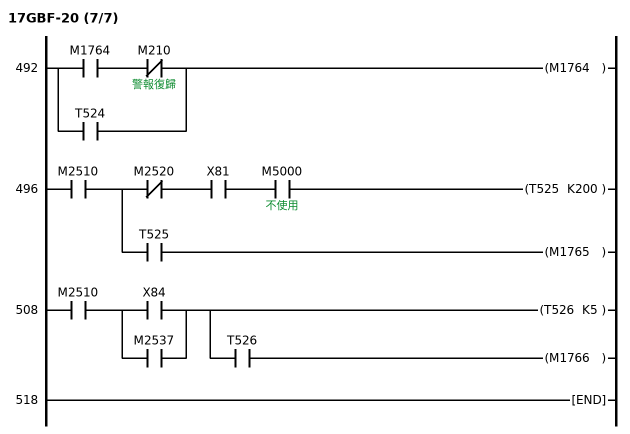
[picture p96: ladder of 17GBF-20, rungs at steps 492 to 518]
492   LD      M1764
      ANI     M210  ; 警報復歸
      OR      T524
      OUT     M1764
496   LD      M2510
      MPS
      ANI     M2520
      AND     X81
      AND     M5000  ; 不使用
      OUT     T525 K200
      MPP
      AND     T525
      OUT     M1765
508   LD      M2510
      LD      X84
      OR      M2537
      ANB
      OUT     T526 K5
      AND     T526
      OUT     M1766
518   END
END_PROGRAM

PROGRAM 18GCV
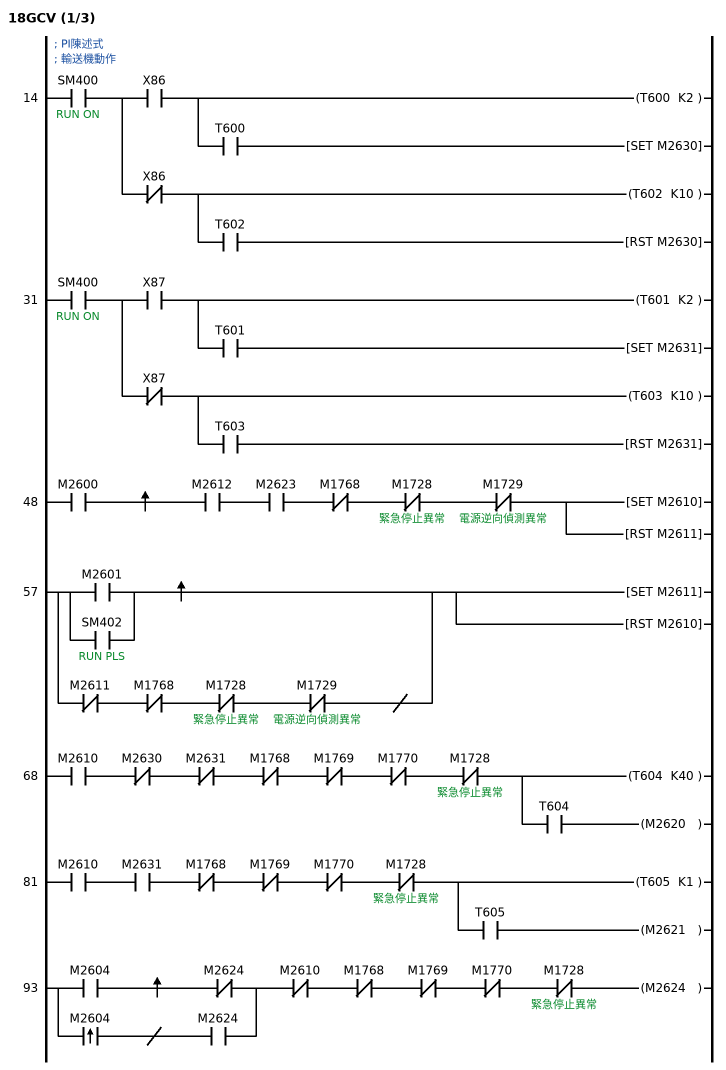
; PI陳述式
; 輸送機動作
14    LD      SM400  ; RUN ON
      MPS
      AND     X86
      OUT     T600 K2
      AND     T600
      SET     M2630
      MPP
      ANI     X86
      OUT     T602 K10
      AND     T602
      RST     M2630
31    LD      SM400  ; RUN ON
      MPS
      AND     X87
      OUT     T601 K2
      AND     T601
      SET     M2631
      MPP
      ANI     X87
      OUT     T603 K10
      AND     T603
      RST     M2631
48    LD      M2600
      MEP
      AND     M2612
      AND     M2623
      ANI     M1768
      ANI     M1728  ; 緊急停止異常
      ANI     M1729  ; 電源逆向偵測異常
      SET     M2610
      RST     M2611
57    LD      M2601
      OR      SM402  ; RUN PLS
      MEP
      LDI     M2611
      ANI     M1768
      ANI     M1728  ; 緊急停止異常
      ANI     M1729  ; 電源逆向偵測異常
      INV
      ORB
      SET     M2611
      RST     M2610
68    LD      M2610
      ANI     M2630
      ANI     M2631
      ANI     M1768
      ANI     M1769
      ANI     M1770
      ANI     M1728  ; 緊急停止異常
      OUT     T604 K40
      AND     T604
      OUT     M2620
81    LD      M2610
      AND     M2631
      ANI     M1768
      ANI     M1769
      ANI     M1770
      ANI     M1728  ; 緊急停止異常
      OUT     T605 K1
      AND     T605
      OUT     M2621
93    LD      M2604
      MEP
      ANI     M2624
      LDP     M2604
      INV
      AND     M2624
      ORB
      ANI     M2610
      ANI     M1768
      ANI     M1769
      ANI     M1770
      ANI     M1728  ; 緊急停止異常
      OUT     M2624
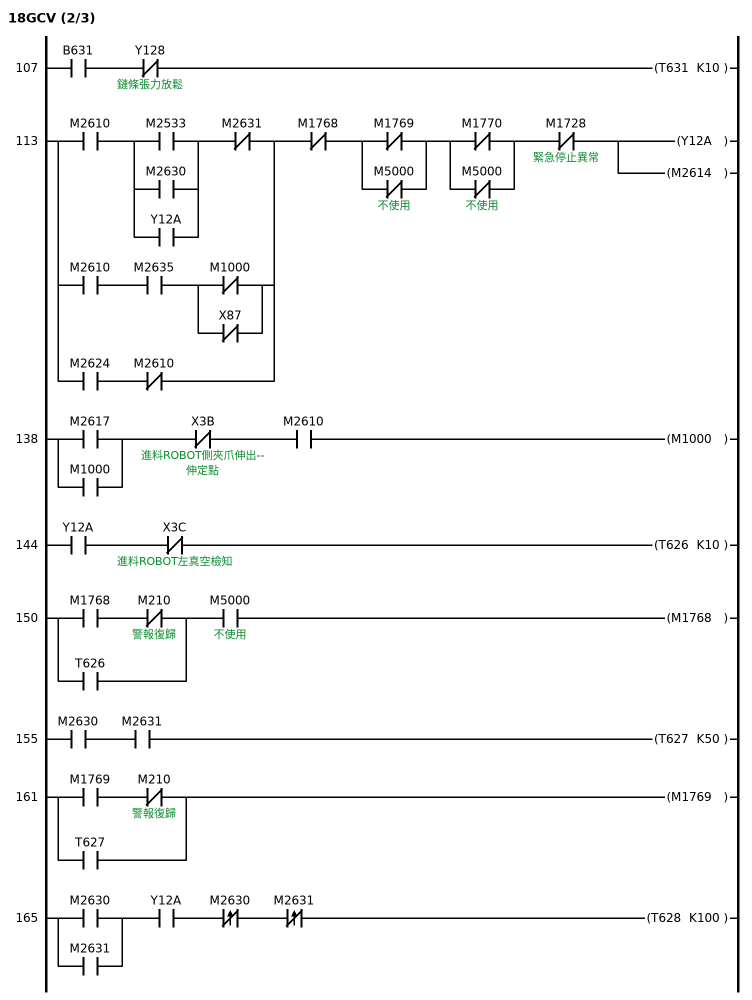
107   LD      B631
      ANI     Y128  ; 鏈條張力放鬆
      OUT     T631 K10
113   LD      M2610
      LD      M2533
      OR      M2630
      OR      Y12A
      ANB
      ANI     M2631
      LD      M2610
      AND     M2635
      LDI     M1000
      ORI     X87
      ANB
      ORB
      LD      M2624
      ANI     M2610
      ORB
      ANI     M1768
      LDI     M1769
      ORI     M5000  ; 不使用
      ANB
      LDI     M1770
      ORI     M5000  ; 不使用
      ANB
      ANI     M1728  ; 緊急停止異常
      OUT     Y12A
      OUT     M2614
138   LD      M2617
      OR      M1000
      ANI     X3B  ; 進料ROBOT側夾爪伸出--伸定點
      AND     M2610
      OUT     M1000
144   LD      Y12A
      ANI     X3C  ; 進料ROBOT左真空檢知
      OUT     T626 K10
150   LD      M1768
      ANI     M210  ; 警報復歸
      OR      T626
      AND     M5000  ; 不使用
      OUT     M1768
155   LD      M2630
      AND     M2631
      OUT     T627 K50
161   LD      M1769
      ANI     M210  ; 警報復歸
      OR      T627
      OUT     M1769
165   LD      M2630
      OR      M2631
      AND     Y12A
      ANDPI   M2630
      ANDPI   M2631
      OUT     T628 K100
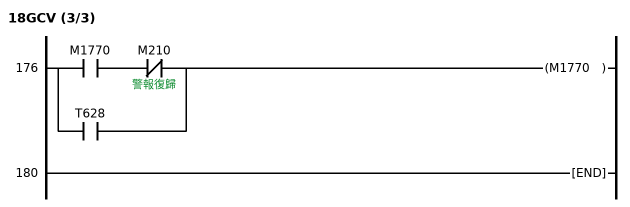
176   LD      M1770
      ANI     M210  ; 警報復歸
      OR      T628
      OUT     M1770
180   END
END_PROGRAM

PROGRAM 19GTC-7
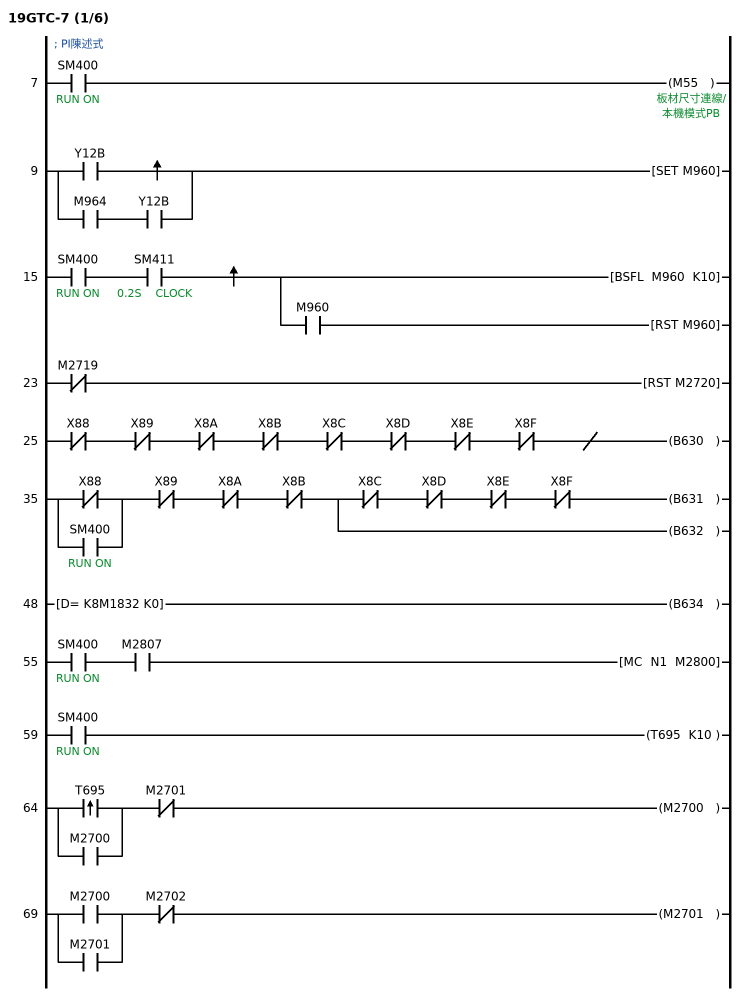
; PI陳述式
7     LD      SM400  ; RUN ON
      OUT     M55  ; 板材尺寸連線/本機模式PB
9     LD      Y12B
      MEP
      LD      M964
      AND     Y12B
      ORB
      SET     M960
15    LD      SM400  ; RUN ON
      AND     SM411  ; 0.2S    CLOCK
      MEP
      BSFL    M960 K10
      AND     M960
      RST     M960
23    LDI     M2719
      RST     M2720
25    LDI     X88
      ANI     X89
      ANI     X8A
      ANI     X8B
      ANI     X8C
      ANI     X8D
      ANI     X8E
      ANI     X8F
      INV
      OUT     B630
35    LDI     X88
      OR      SM400  ; RUN ON
      ANI     X89
      ANI     X8A
      ANI     X8B
      MPS
      ANI     X8C
      ANI     X8D
      ANI     X8E
      ANI     X8F
      OUT     B631
      MPP
      OUT     B632
48    LDD=    K8M1832 K0
      OUT     B634
55    LD      SM400  ; RUN ON
      AND     M2807
      MC      N1 M2800
59    LD      SM400  ; RUN ON
      OUT     T695 K10
64    LDP     T695
      OR      M2700
      ANI     M2701
      OUT     M2700
69    LD      M2700
      OR      M2701
      ANI     M2702
      OUT     M2701
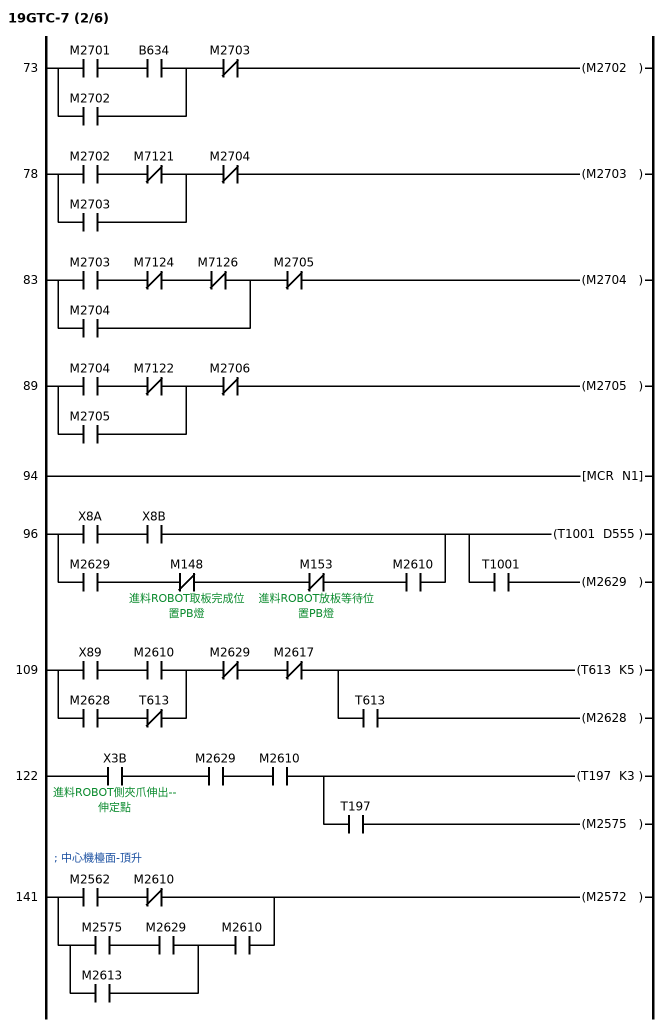
73    LD      M2701
      AND     B634
      OR      M2702
      ANI     M2703
      OUT     M2702
78    LD      M2702
      ANI     M7121
      OR      M2703
      ANI     M2704
      OUT     M2703
83    LD      M2703
      ANI     M7124
      ANI     M7126
      OR      M2704
      ANI     M2705
      OUT     M2704
89    LD      M2704
      ANI     M7122
      OR      M2705
      ANI     M2706
      OUT     M2705
94    MCR     N1
96    LD      X8A
      AND     X8B
      LD      M2629
      ANI     M148  ; 進料ROBOT取板完成位置PB燈
      ANI     M153  ; 進料ROBOT放板等待位置PB燈
      AND     M2610
      ORB
      OUT     T1001 D555
      AND     T1001
      OUT     M2629
109   LD      X89
      AND     M2610
      LD      M2628
      ANI     T613
      ORB
      ANI     M2629
      ANI     M2617
      OUT     T613 K5
      AND     T613
      OUT     M2628
122   LD      X3B  ; 進料ROBOT側夾爪伸出--伸定點
      AND     M2629
      AND     M2610
      OUT     T197 K3
      AND     T197
      OUT     M2575
; 中心機檯面-頂升
141   LD      M2562
      ANI     M2610
      LD      M2575
      AND     M2629
      OR      M2613
      AND     M2610
      ORB
      OUT     M2572
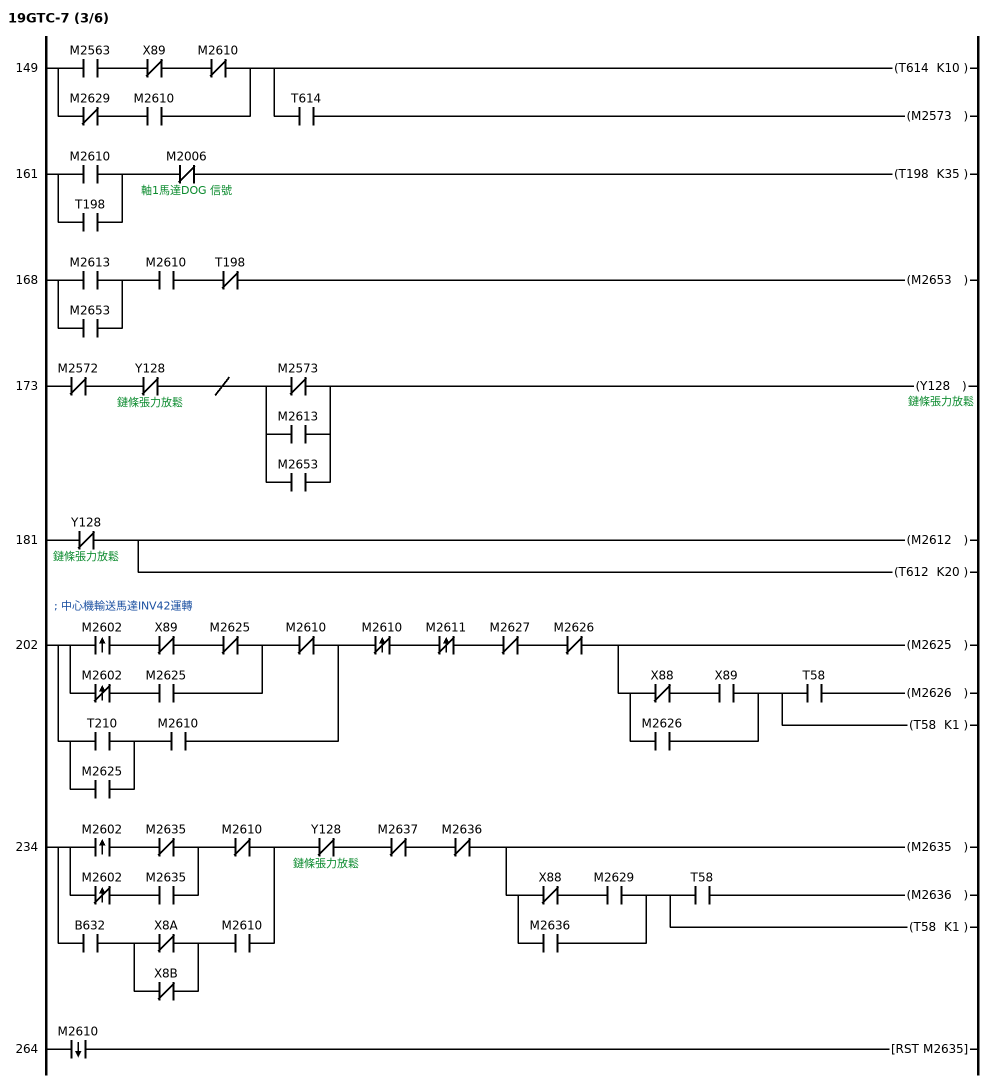
149   LD      M2563
      ANI     X89
      ANI     M2610
      LDI     M2629
      AND     M2610
      ORB
      OUT     T614 K10
      AND     T614
      OUT     M2573
161   LD      M2610
      OR      T198
      ANI     M2006  ; 軸1馬達DOG 信號
      OUT     T198 K35
168   LD      M2613
      OR      M2653
      AND     M2610
      ANI     T198
      OUT     M2653
173   LDI     M2572
      ANI     Y128  ; 鏈條張力放鬆
      INV
      LDI     M2573
      OR      M2613
      OR      M2653
      ANB
      OUT     Y128  ; 鏈條張力放鬆
181   LDI     Y128  ; 鏈條張力放鬆
      OUT     M2612
      OUT     T612 K20
; 中心機輸送馬達INV42運轉
202   LDP     M2602
      ANI     X89
      ANI     M2625
      LDPI    M2602
      AND     M2625
      ORB
      ANI     M2610
      LD      T210
      OR      M2625
      AND     M2610
      ORB
      ANDPI   M2610
      ANDPI   M2611
      ANI     M2627
      ANI     M2626
      OUT     M2625
      LDI     X88
      AND     X89
      OR      M2626
      ANB
      MPS
      AND     T58
      OUT     M2626
      MPP
      OUT     T58 K1
234   LDP     M2602
      ANI     M2635
      LDPI    M2602
      AND     M2635
      ORB
      ANI     M2610
      LD      B632
      LDI     X8A
      ORI     X8B
      ANB
      AND     M2610
      ORB
      ANI     Y128  ; 鏈條張力放鬆
      ANI     M2637
      ANI     M2636
      OUT     M2635
      LDI     X88
      AND     M2629
      OR      M2636
      ANB
      MPS
      AND     T58
      OUT     M2636
      MPP
      OUT     T58 K1
264   LDF     M2610
      RST     M2635
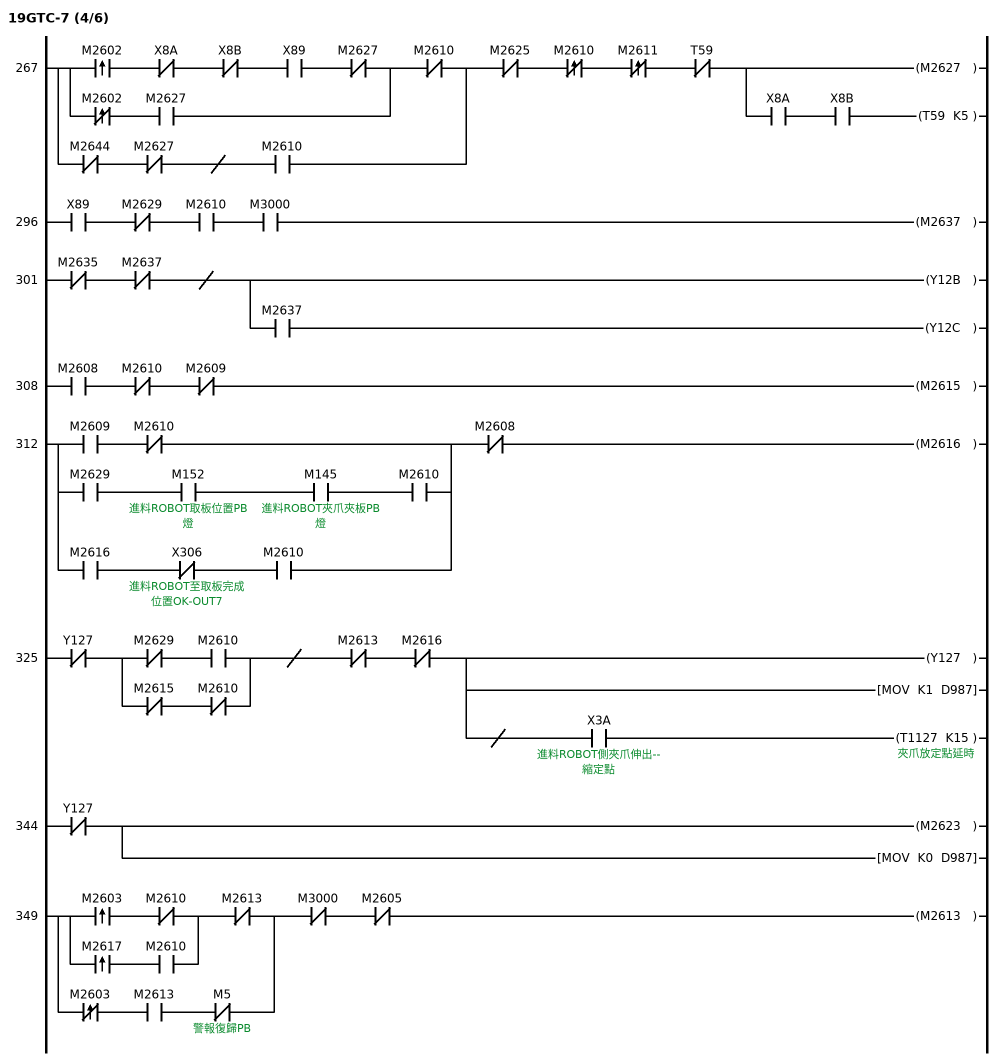
267   LDP     M2602
      ANI     X8A
      ANI     X8B
      AND     X89
      ANI     M2627
      LDPI    M2602
      AND     M2627
      ORB
      ANI     M2610
      LDI     M2644
      ANI     M2627
      INV
      AND     M2610
      ORB
      ANI     M2625
      ANDPI   M2610
      ANDPI   M2611
      ANI     T59
      OUT     M2627
      AND     X8A
      AND     X8B
      OUT     T59 K5
296   LD      X89
      ANI     M2629
      AND     M2610
      AND     M3000
      OUT     M2637
301   LDI     M2635
      ANI     M2637
      INV
      OUT     Y12B
      AND     M2637
      OUT     Y12C
308   LD      M2608
      ANI     M2610
      ANI     M2609
      OUT     M2615
312   LD      M2609
      ANI     M2610
      LD      M2629
      AND     M152  ; 進料ROBOT取板位置PB燈
      AND     M145  ; 進料ROBOT夾爪夾板PB燈
      AND     M2610
      ORB
      LD      M2616
      ANI     X306  ; 進料ROBOT至取板完成位置OK-OUT7
      AND     M2610
      ORB
      ANI     M2608
      OUT     M2616
325   LDI     Y127
      LDI     M2629
      AND     M2610
      LDI     M2615
      ANI     M2610
      ORB
      ANB
      INV
      ANI     M2613
      ANI     M2616
      OUT     Y127
      MOV     K1 D987
      INV
      AND     X3A  ; 進料ROBOT側夾爪伸出--縮定點
      OUT     T1127 K15  ; 夾爪放定點延時
344   LDI     Y127
      OUT     M2623
      MOV     K0 D987
349   LDP     M2603
      ANI     M2610
      LDP     M2617
      AND     M2610
      ORB
      ANI     M2613
      LDPI    M2603
      AND     M2613
      ANI     M5  ; 警報復歸PB
      ORB
      ANI     M3000
      ANI     M2605
      OUT     M2613
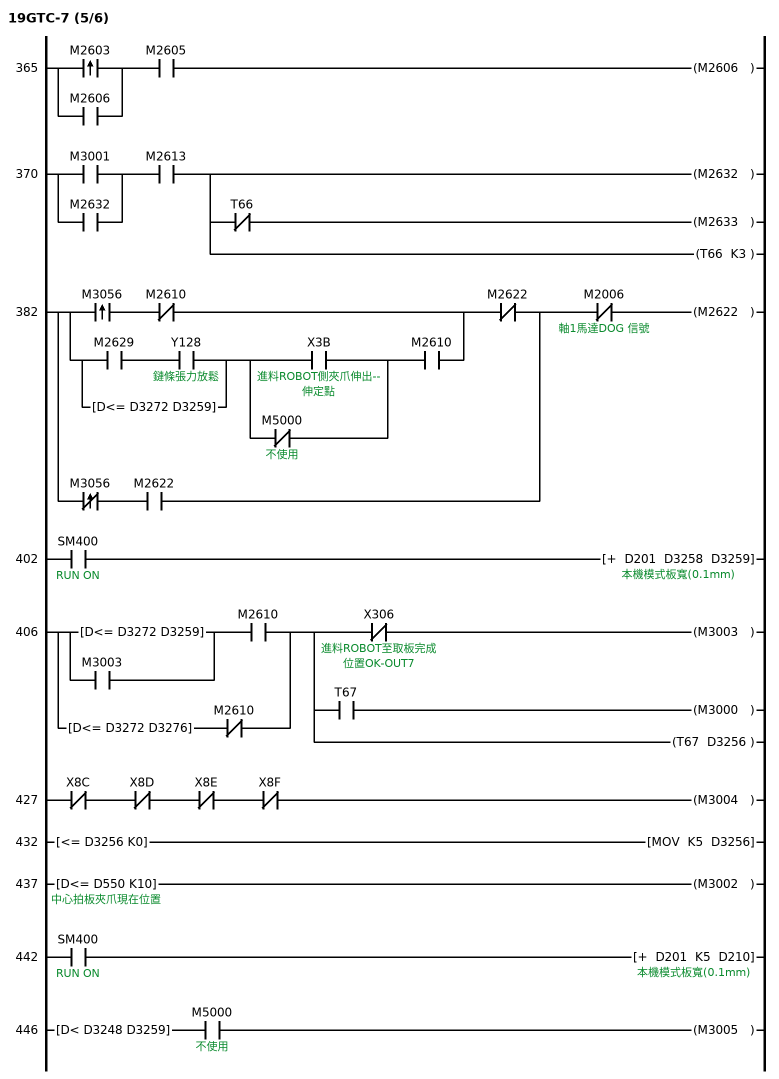
365   LDP     M2603
      OR      M2606
      AND     M2605
      OUT     M2606
370   LD      M3001
      OR      M2632
      AND     M2613
      OUT     M2632
      MPS
      ANI     T66
      OUT     M2633
      MPP
      OUT     T66 K3
382   LDP     M3056
      ANI     M2610
      LD      M2629
      AND     Y128  ; 鏈條張力放鬆
      ORD<=   D3272 D3259
      LD      X3B  ; 進料ROBOT側夾爪伸出--伸定點
      ORI     M5000  ; 不使用
      ANB
      AND     M2610
      ORB
      ANI     M2622
      LDPI    M3056
      AND     M2622
      ORB
      ANI     M2006  ; 軸1馬達DOG 信號
      OUT     M2622
402   LD      SM400  ; RUN ON
      +       D201 D3258 D3259  ; 本機模式板寬(0.1mm)
406   LDD<=   D3272 D3259
      OR      M3003
      AND     M2610
      LDD<=   D3272 D3276
      ANI     M2610
      ORB
      MPS
      ANI     X306  ; 進料ROBOT至取板完成位置OK-OUT7
      OUT     M3003
      MRD
      AND     T67
      OUT     M3000
      MPP
      OUT     T67 D3256
427   LDI     X8C
      ANI     X8D
      ANI     X8E
      ANI     X8F
      OUT     M3004
432   LD<=    D3256 K0
      MOV     K5 D3256
437   LDD<=   D550 K10  ; 中心拍板夾爪現在位置
      OUT     M3002
442   LD      SM400  ; RUN ON
      +       D201 K5 D210
446   LDD<    D3248 D3259
      AND     M5000  ; 不使用
      OUT     M3005
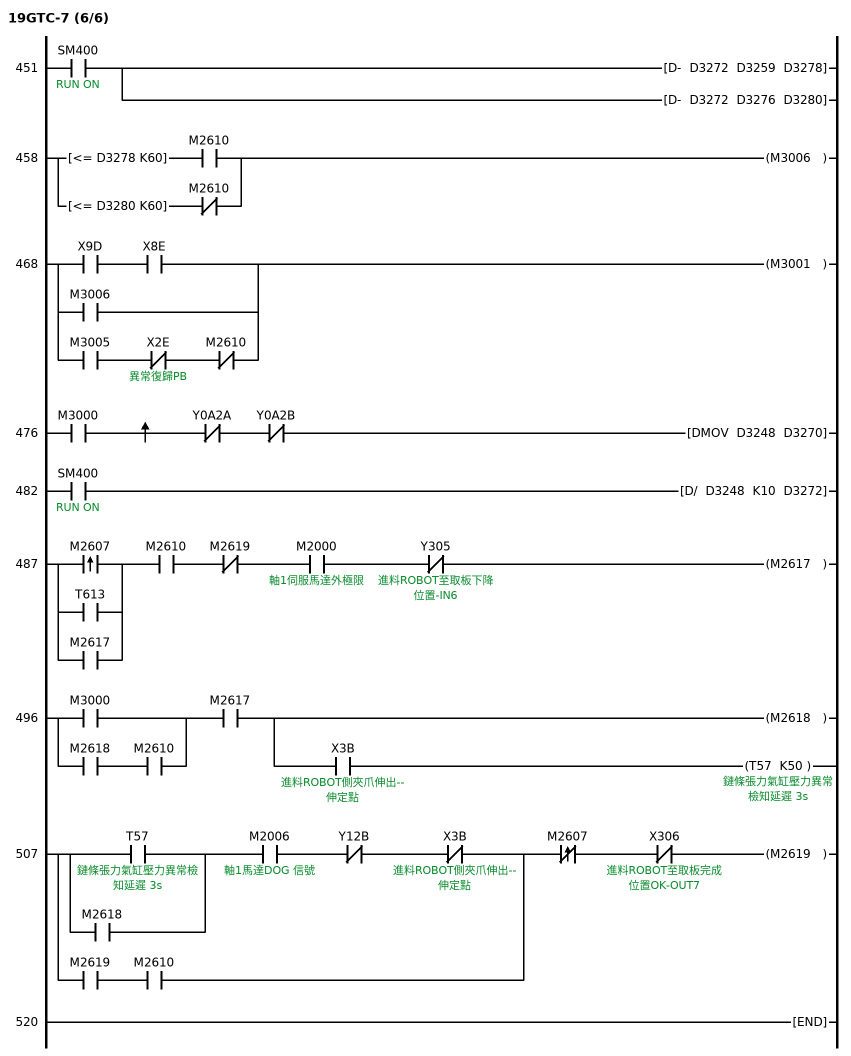
451   LD      SM400  ; RUN ON
      D-      D3272 D3259 D3278
      D-      D3272 D3276 D3280
458   LD<=    D3278 K60
      AND     M2610
      LD<=    D3280 K60
      ANI     M2610
      ORB
      OUT     M3006
468   LD      X9D
      AND     X8E
      OR      M3006
      LD      M3005
      ANI     X2E  ; 異常復歸PB
      ANI     M2610
      ORB
      OUT     M3001
476   LD      M3000
      MEP
      ANI     Y0A2A
      ANI     Y0A2B
      DMOV    D3248 D3270
482   LD      SM400  ; RUN ON
      D/      D3248 K10 D3272
487   LDP     M2607
      OR      T613
      OR      M2617
      AND     M2610
      ANI     M2619
      AND     M2000  ; 軸1伺服馬達外極限
      ANI     Y305  ; 進料ROBOT至取板下降位置-IN6
      OUT     M2617
496   LD      M3000
      LD      M2618
      AND     M2610
      ORB
      AND     M2617
      OUT     M2618
      AND     X3B  ; 進料ROBOT側夾爪伸出--伸定點
      OUT     T57 K50  ; 鏈條張力氣缸壓力異常檢知延遲 3s
507   LD      T57  ; 鏈條張力氣缸壓力異常檢知延遲 3s
      OR      M2618
      AND     M2006  ; 軸1馬達DOG 信號
      ANI     Y12B
      ANI     X3B  ; 進料ROBOT側夾爪伸出--伸定點
      LD      M2619
      AND     M2610
      ORB
      ANDPI   M2607
      ANI     X306  ; 進料ROBOT至取板完成位置OK-OUT7
      OUT     M2619
520   END
END_PROGRAM

PROGRAM 20TEST
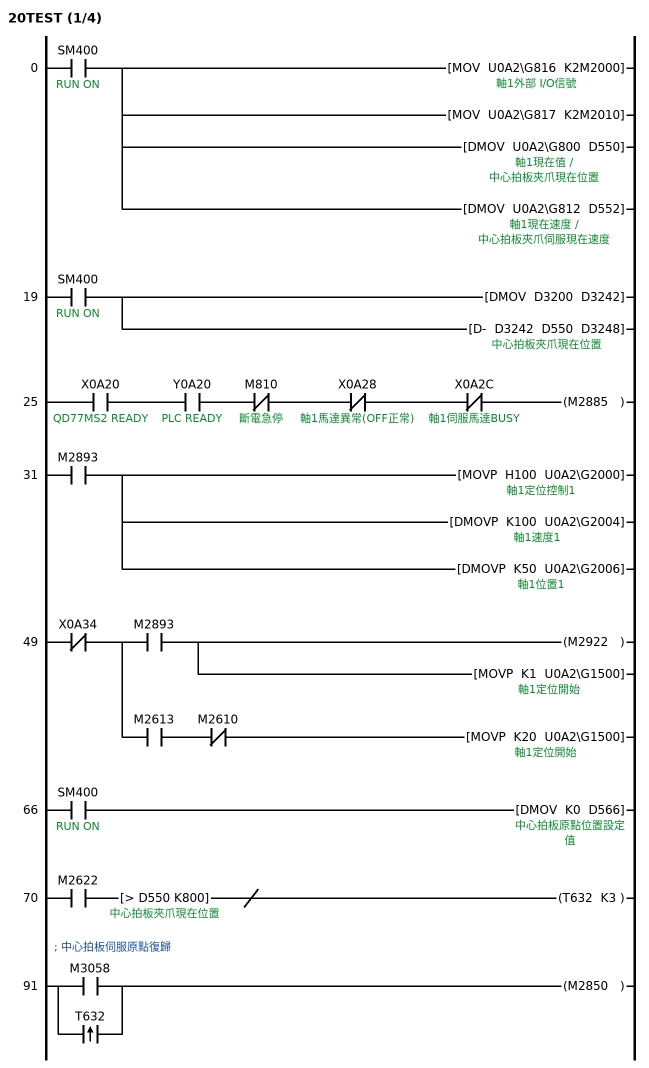
0     LD      SM400  ; RUN ON
      MOV     U0A2\G816 K2M2000  ; 軸1外部 I/O信號 / 軸1伺服馬達外極限
      MOV     U0A2\G817 K2M2010
      DMOV    U0A2\G800 D550  ; 軸1現在值 / 中心拍板夾爪現在位置
      DMOV    U0A2\G812 D552  ; 軸1現在速度 / 中心拍板夾爪伺服現在速度
19    LD      SM400  ; RUN ON
      DMOV    D3200 D3242
      D-      D3242 D550 D3248
25    LD      X0A20  ; QD77MS2 READY
      AND     Y0A20  ; PLC READY
      ANI     M810  ; 斷電急停
      ANI     X0A28  ; 軸1馬達異常(OFF正常)
      ANI     X0A2C  ; 軸1伺服馬達BUSY
      OUT     M2885
31    LD      M2893
      MOVP    H100 U0A2\G2000  ; 軸1定位控制1
      DMOVP   K100 U0A2\G2004  ; 軸1速度1
      DMOVP   K50 U0A2\G2006  ; 軸1位置1
49    LDI     X0A34
      MPS
      AND     M2893
      OUT     M2922
      MOVP    K1 U0A2\G1500  ; 軸1定位開始
      MPP
      AND     M2613
      ANI     M2610
      MOVP    K20 U0A2\G1500
66    LD      SM400  ; RUN ON
      DMOV    K0 D566  ; 中心拍板原點位置設定值
70    LD      M2622
      AND>    D550 K800  ; 中心拍板夾爪現在位置
      INV
      OUT     T632 K3
; 中心拍板伺服原點復歸
91    LD      M3058
      ORP     T632
      OUT     M2850
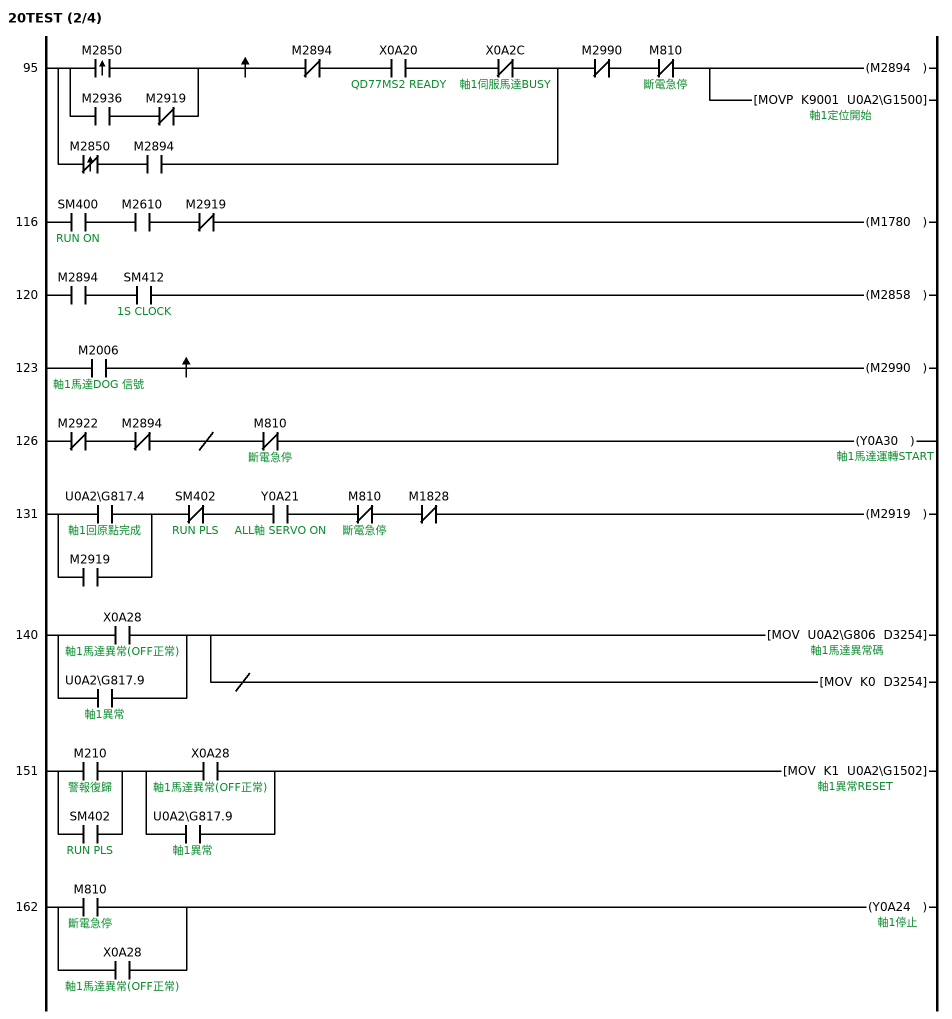
95    LDP     M2850
      LD      M2936
      ANI     M2919
      ORB
      MEP
      ANI     M2894
      AND     X0A20  ; QD77MS2 READY
      ANI     X0A2C  ; 軸1伺服馬達BUSY
      LDPI    M2850
      AND     M2894
      ORB
      ANI     M2990
      ANI     M810  ; 斷電急停
      OUT     M2894
      MOVP    K9001 U0A2\G1500
116   LD      SM400  ; RUN ON
      AND     M2610
      ANI     M2919
      OUT     M1780
120   LD      M2894
      AND     SM412  ; 1S CLOCK
      OUT     M2858
123   LD      M2006  ; 軸1馬達DOG 信號
      MEP
      OUT     M2990
126   LDI     M2922
      ANI     M2894
      INV
      ANI     M810  ; 斷電急停
      OUT     Y0A30  ; 軸1馬達運轉START
131   LD      U0A2\G817.4  ; 軸1回原點完成
      OR      M2919
      ANI     SM402  ; RUN PLS
      AND     Y0A21  ; ALL軸 SERVO ON
      ANI     M810  ; 斷電急停
      ANI     M1828
      OUT     M2919
140   LD      X0A28  ; 軸1馬達異常(OFF正常)
      OR      U0A2\G817.9  ; 軸1異常
      MOV     U0A2\G806 D3254  ; 軸1馬達異常碼
      INV
      MOV     K0 D3254
151   LD      M210  ; 警報復歸
      OR      SM402  ; RUN PLS
      LD      X0A28  ; 軸1馬達異常(OFF正常)
      OR      U0A2\G817.9  ; 軸1異常
      ANB
      MOV     K1 U0A2\G1502  ; 軸1異常RESET
162   LD      M810  ; 斷電急停
      OR      X0A28  ; 軸1馬達異常(OFF正常)
      OUT     Y0A24  ; 軸1停止
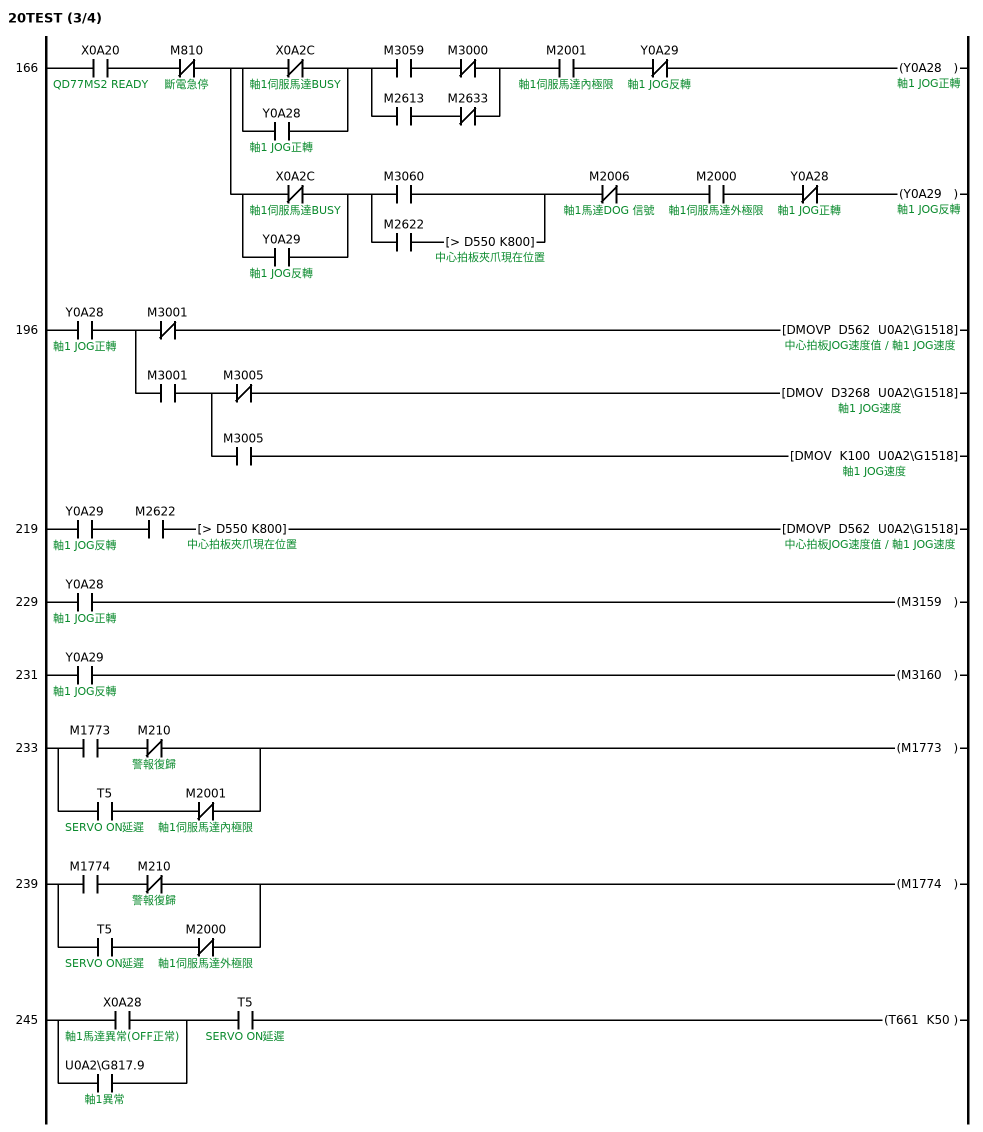
166   LD      X0A20  ; QD77MS2 READY
      ANI     M810  ; 斷電急停
      MPS
      LDI     X0A2C  ; 軸1伺服馬達BUSY
      OR      Y0A28  ; 軸1 JOG正轉
      ANB
      LD      M3059
      ANI     M3000
      LD      M2613
      ANI     M2633
      ORB
      ANB
      AND     M2001  ; 軸1伺服馬達內極限
      ANI     Y0A29  ; 軸1 JOG反轉
      OUT     Y0A28  ; 軸1 JOG正轉
      MPP
      LDI     X0A2C  ; 軸1伺服馬達BUSY
      OR      Y0A29  ; 軸1 JOG反轉
      ANB
      LD      M3060
      LD      M2622
      AND>    D550 K800  ; 中心拍板夾爪現在位置
      ORB
      ANB
      ANI     M2006  ; 軸1馬達DOG 信號
      AND     M2000  ; 軸1伺服馬達外極限
      ANI     Y0A28  ; 軸1 JOG正轉
      OUT     Y0A29  ; 軸1 JOG反轉
196   LD      Y0A28  ; 軸1 JOG正轉
      MPS
      ANI     M3001
      DMOVP   D562 U0A2\G1518  ; 中心拍板JOG速度值 / 軸1 JOG速度
      MPP
      AND     M3001
      MPS
      ANI     M3005
      DMOV    D3268 U0A2\G1518
      MPP
      AND     M3005
      DMOV    K100 U0A2\G1518
219   LD      Y0A29  ; 軸1 JOG反轉
      AND     M2622
      AND>    D550 K800  ; 中心拍板夾爪現在位置
      DMOVP   D562 U0A2\G1518
229   LD      Y0A28  ; 軸1 JOG正轉
      OUT     M3159
231   LD      Y0A29  ; 軸1 JOG反轉
      OUT     M3160
233   LD      M1773
      ANI     M210  ; 警報復歸
      LD      T5  ; SERVO ON延遲
      ANI     M2001  ; 軸1伺服馬達內極限
      ORB
      OUT     M1773
239   LD      M1774
      ANI     M210  ; 警報復歸
      LD      T5  ; SERVO ON延遲
      ANI     M2000  ; 軸1伺服馬達外極限
      ORB
      OUT     M1774
245   LD      X0A28  ; 軸1馬達異常(OFF正常)
      OR      U0A2\G817.9  ; 軸1異常
      AND     T5  ; SERVO ON延遲
      OUT     T661 K50
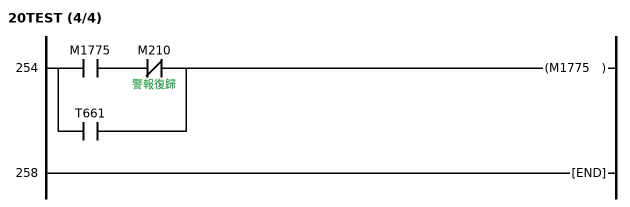
254   LD      M1775
      ANI     M210  ; 警報復歸
      OR      T661
      OUT     M1775
258   END
END_PROGRAM

PROGRAM 21CIM
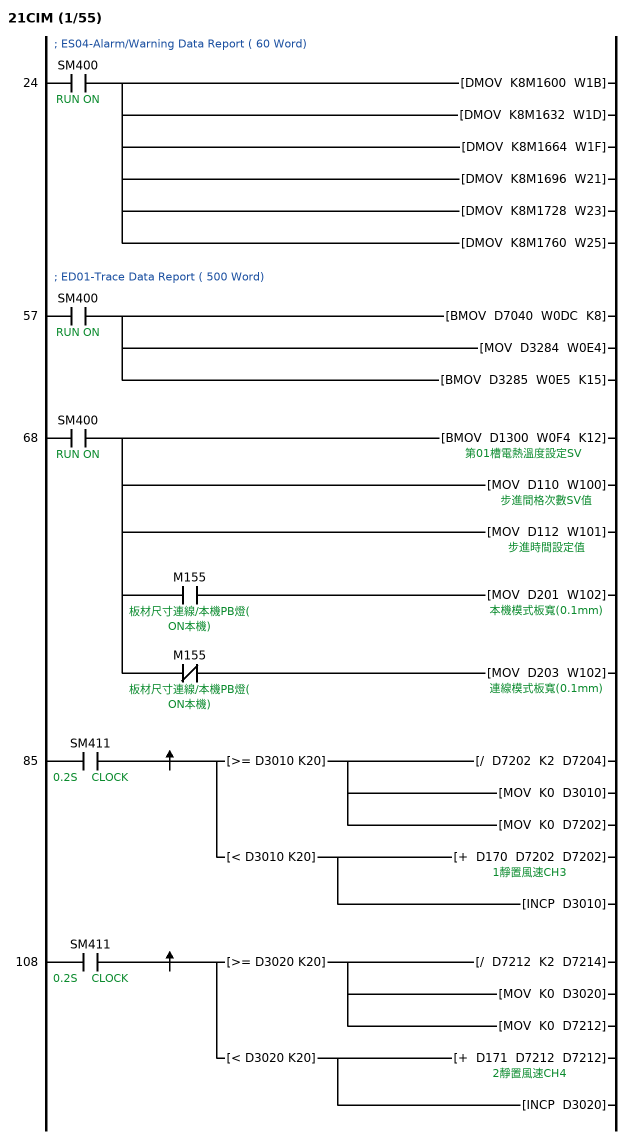
; ES04-Alarm/Warning Data Report ( 60 Word)
24    LD      SM400  ; RUN ON
      DMOV    K8M1600 W1B  ; #01 電熱AL2 超溫
      DMOV    K8M1632 W1D  ; #01 風車過載
      DMOV    K8M1664 W1F  ; 進料風車過載異常
      DMOV    K8M1696 W21  ; 進料夾爪開異常
      DMOV    K8M1728 W23  ; 緊急停止異常
      DMOV    K8M1760 W25
; ED01-Trace Data Report ( 500 Word)
57    LD      SM400  ; RUN ON
      BMOV    D7040 W0DC K8
      MOV     D3284 W0E4
      BMOV    D3285 W0E5 K15
68    LD      SM400  ; RUN ON
      BMOV    D1300 W0F4 K12  ; 第01槽電熱溫度設定SV
      MOV     D110 W100  ; 步進間格次數SV值
      MOV     D112 W101  ; 步進時間設定值
      MPS
      AND     M155  ; 板材尺寸連線/本機PB燈(ON本機)
      MOV     D201 W102  ; 本機模式板寬(0.1mm)
      MPP
      ANI     M155  ; 板材尺寸連線/本機PB燈(ON本機)
      MOV     D203 W102  ; 連線模式板寬(0.1mm)
85    LD      SM411  ; 0.2S    CLOCK
      MEP
      MPS
      AND>=   D3010 K20
      /       D7202 K2 D7204
      MOV     K0 D3010
      MOV     K0 D7202
      MPP
      AND<    D3010 K20
      +       D170 D7202 D7202  ; 1靜置風速CH3
      INCP    D3010
108   LD      SM411  ; 0.2S    CLOCK
      MEP
      MPS
      AND>=   D3020 K20
      /       D7212 K2 D7214
      MOV     K0 D3020
      MOV     K0 D7212
      MPP
      AND<    D3020 K20
      +       D171 D7212 D7212  ; 2靜置風速CH4
      INCP    D3020
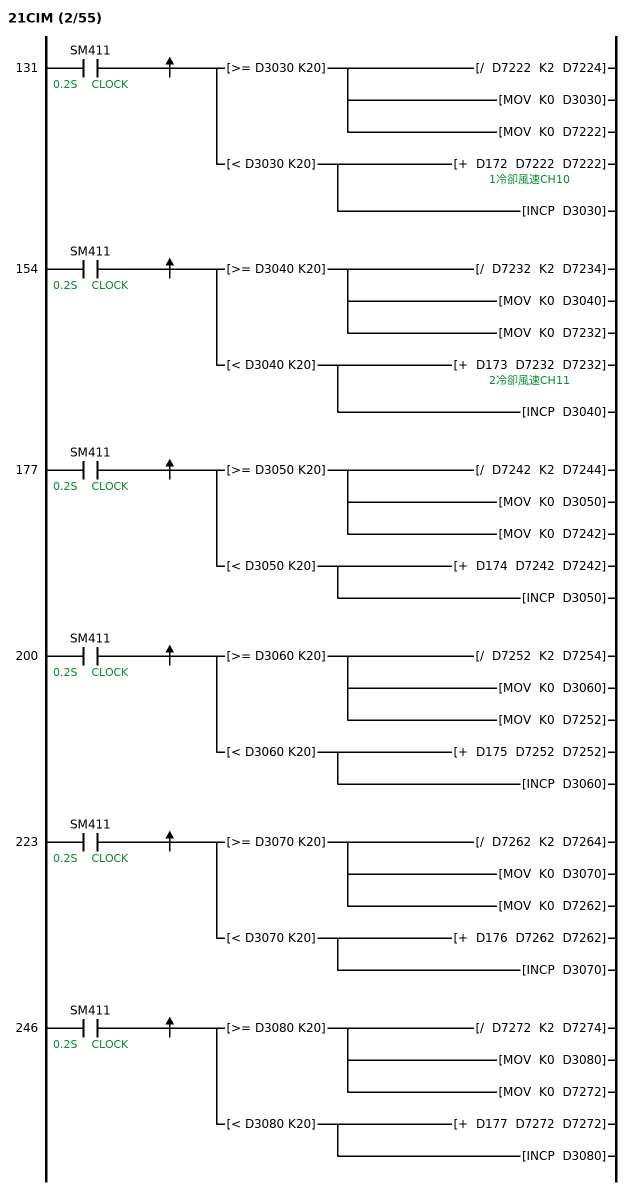
131   LD      SM411  ; 0.2S    CLOCK
      MEP
      MPS
      AND>=   D3030 K20
      /       D7222 K2 D7224
      MOV     K0 D3030
      MOV     K0 D7222
      MPP
      AND<    D3030 K20
      +       D172 D7222 D7222  ; 1冷卻風速CH10
      INCP    D3030
154   LD      SM411  ; 0.2S    CLOCK
      MEP
      MPS
      AND>=   D3040 K20
      /       D7232 K2 D7234
      MOV     K0 D3040
      MOV     K0 D7232
      MPP
      AND<    D3040 K20
      +       D173 D7232 D7232  ; 2冷卻風速CH11
      INCP    D3040
177   LD      SM411  ; 0.2S    CLOCK
      MEP
      MPS
      AND>=   D3050 K20
      /       D7242 K2 D7244
      MOV     K0 D3050
      MOV     K0 D7242
      MPP
      AND<    D3050 K20
      +       D174 D7242 D7242
      INCP    D3050
200   LD      SM411  ; 0.2S    CLOCK
      MEP
      MPS
      AND>=   D3060 K20
      /       D7252 K2 D7254
      MOV     K0 D3060
      MOV     K0 D7252
      MPP
      AND<    D3060 K20
      +       D175 D7252 D7252
      INCP    D3060
223   LD      SM411  ; 0.2S    CLOCK
      MEP
      MPS
      AND>=   D3070 K20
      /       D7262 K2 D7264
      MOV     K0 D3070
      MOV     K0 D7262
      MPP
      AND<    D3070 K20
      +       D176 D7262 D7262
      INCP    D3070
246   LD      SM411  ; 0.2S    CLOCK
      MEP
      MPS
      AND>=   D3080 K20
      /       D7272 K2 D7274
      MOV     K0 D3080
      MOV     K0 D7272
      MPP
      AND<    D3080 K20
      +       D177 D7272 D7272
      INCP    D3080
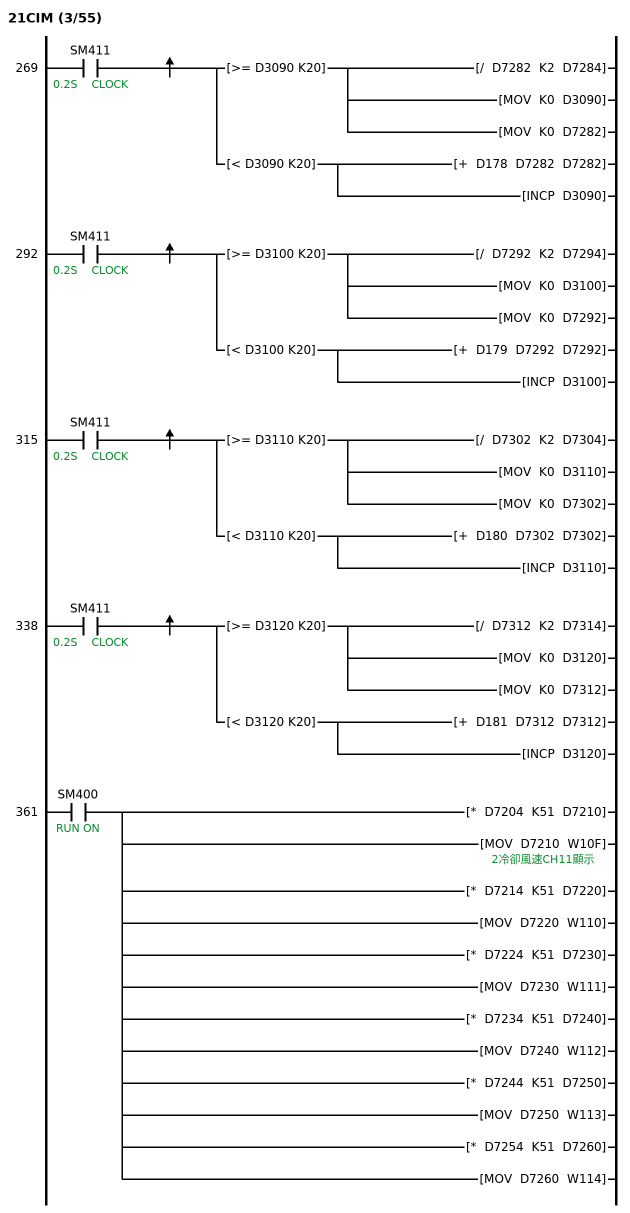
269   LD      SM411  ; 0.2S    CLOCK
      MEP
      MPS
      AND>=   D3090 K20
      /       D7282 K2 D7284
      MOV     K0 D3090
      MOV     K0 D7282
      MPP
      AND<    D3090 K20
      +       D178 D7282 D7282
      INCP    D3090
292   LD      SM411  ; 0.2S    CLOCK
      MEP
      MPS
      AND>=   D3100 K20
      /       D7292 K2 D7294
      MOV     K0 D3100
      MOV     K0 D7292
      MPP
      AND<    D3100 K20
      +       D179 D7292 D7292
      INCP    D3100
315   LD      SM411  ; 0.2S    CLOCK
      MEP
      MPS
      AND>=   D3110 K20
      /       D7302 K2 D7304
      MOV     K0 D3110
      MOV     K0 D7302
      MPP
      AND<    D3110 K20
      +       D180 D7302 D7302
      INCP    D3110
338   LD      SM411  ; 0.2S    CLOCK
      MEP
      MPS
      AND>=   D3120 K20
      /       D7312 K2 D7314
      MOV     K0 D3120
      MOV     K0 D7312
      MPP
      AND<    D3120 K20
      +       D181 D7312 D7312
      INCP    D3120
361   LD      SM400  ; RUN ON
      *       D7204 K51 D7210
      MOV     D7210 W10F  ; 2冷卻風速CH11顯示
      *       D7214 K51 D7220
      MOV     D7220 W110
      *       D7224 K51 D7230
      MOV     D7230 W111
      *       D7234 K51 D7240
      MOV     D7240 W112
      *       D7244 K51 D7250
      MOV     D7250 W113
      *       D7254 K51 D7260
      MOV     D7260 W114
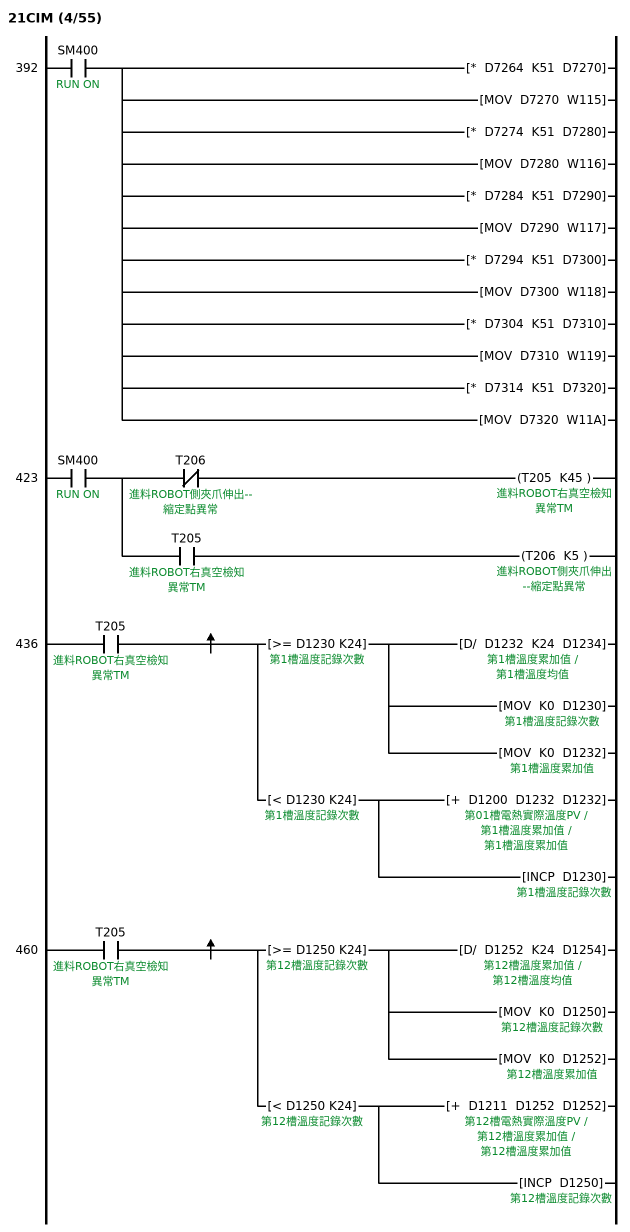
392   LD      SM400  ; RUN ON
      *       D7264 K51 D7270
      MOV     D7270 W115
      *       D7274 K51 D7280
      MOV     D7280 W116
      *       D7284 K51 D7290
      MOV     D7290 W117
      *       D7294 K51 D7300
      MOV     D7300 W118
      *       D7304 K51 D7310
      MOV     D7310 W119
      *       D7314 K51 D7320
      MOV     D7320 W11A
423   LD      SM400  ; RUN ON
      MPS
      ANI     T206  ; 進料ROBOT側夾爪伸出--縮定點異常
      OUT     T205 K45  ; 進料ROBOT右真空檢知異常TM
      MPP
      AND     T205  ; 進料ROBOT右真空檢知異常TM
      OUT     T206 K5  ; 進料ROBOT側夾爪伸出--縮定點異常
436   LD      T205  ; 進料ROBOT右真空檢知異常TM
      MEP
      MPS
      AND>=   D1230 K24  ; 第1槽溫度記錄次數
      D/      D1232 K24 D1234  ; 第1槽溫度累加值 / 第1槽溫度均值
      MOV     K0 D1230
      MOV     K0 D1232
      MPP
      AND<    D1230 K24  ; 第1槽溫度記錄次數
      +       D1200 D1232 D1232  ; 第01槽電熱實際溫度PV
      INCP    D1230
460   LD      T205  ; 進料ROBOT右真空檢知異常TM
      MEP
      MPS
      AND>=   D1250 K24  ; 第12槽溫度記錄次數
      D/      D1252 K24 D1254  ; 第12槽溫度累加值 / 第12槽溫度均值
      MOV     K0 D1250
      MOV     K0 D1252
      MPP
      AND<    D1250 K24  ; 第12槽溫度記錄次數
      +       D1211 D1252 D1252  ; 第12槽電熱實際溫度PV
      INCP    D1250
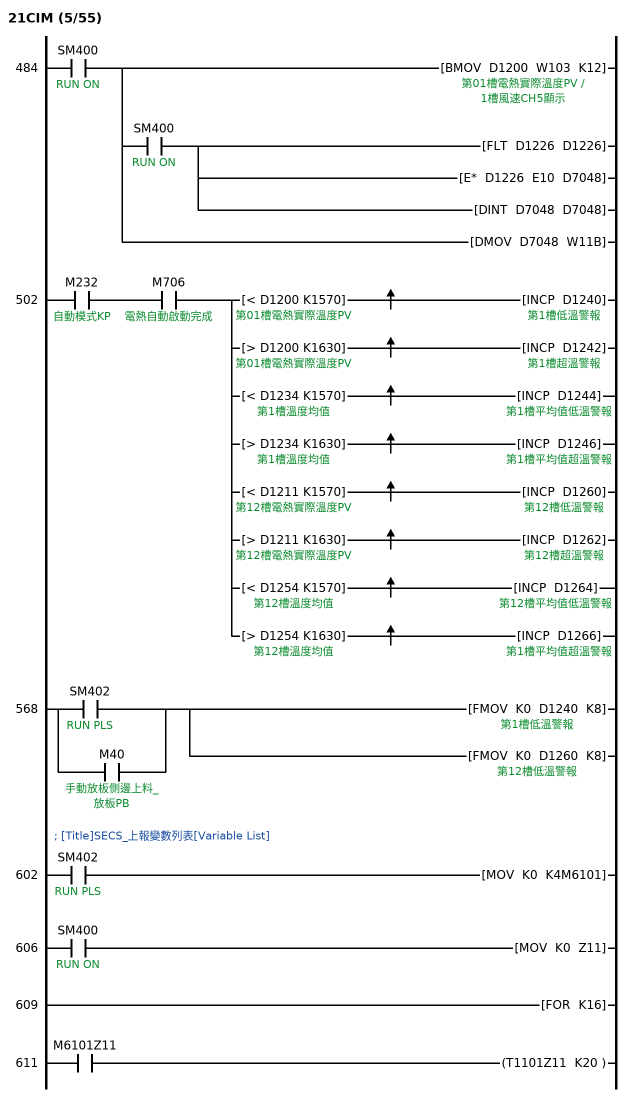
484   LD      SM400  ; RUN ON
      BMOV    D1200 W103 K12  ; 1槽風速CH5顯示
      MPS
      AND     SM400  ; RUN ON
      FLT     D1226 D1226
      E*      D1226 E10 D7048
      DINT    D7048 D7048
      MPP
      DMOV    D7048 W11B
502   LD      M232  ; 自動模式KP
      AND     M706  ; 電熱自動啟動完成
      MPS
      AND<    D1200 K1570  ; 第01槽電熱實際溫度PV
      MEP
      INCP    D1240  ; 第1槽低溫警報
      MRD
      AND>    D1200 K1630  ; 第01槽電熱實際溫度PV
      MEP
      INCP    D1242  ; 第1槽超溫警報
      MRD
      AND<    D1234 K1570  ; 第1槽溫度均值
      MEP
      INCP    D1244  ; 第1槽平均值低溫警報
      MRD
      AND>    D1234 K1630  ; 第1槽溫度均值
      MEP
      INCP    D1246  ; 第1槽平均值超溫警報
      MRD
      AND<    D1211 K1570  ; 第12槽電熱實際溫度PV
      MEP
      INCP    D1260  ; 第12槽低溫警報
      MRD
      AND>    D1211 K1630  ; 第12槽電熱實際溫度PV
      MEP
      INCP    D1262  ; 第12槽超溫警報
      MRD
      AND<    D1254 K1570  ; 第12槽溫度均值
      MEP
      INCP    D1264  ; 第12槽平均值低溫警報
      MPP
      AND>    D1254 K1630  ; 第12槽溫度均值
      MEP
      INCP    D1266  ; 第1槽平均值超溫警報
568   LD      SM402  ; RUN PLS
      OR      M40  ; 手動放板側邊上料_放板PB
      FMOV    K0 D1240 K8
      FMOV    K0 D1260 K8
; [Title]SECS_上報變數列表[Variable List]
602   LD      SM402  ; RUN PLS
      MOV     K0 K4M6101  ; EQP->SES控制模式切換(Online/Off)
606   LD      SM400  ; RUN ON
      MOV     K0 Z11
609   FOR     K16
611   LD      M6101Z11
      OUT     T1101Z11 K20
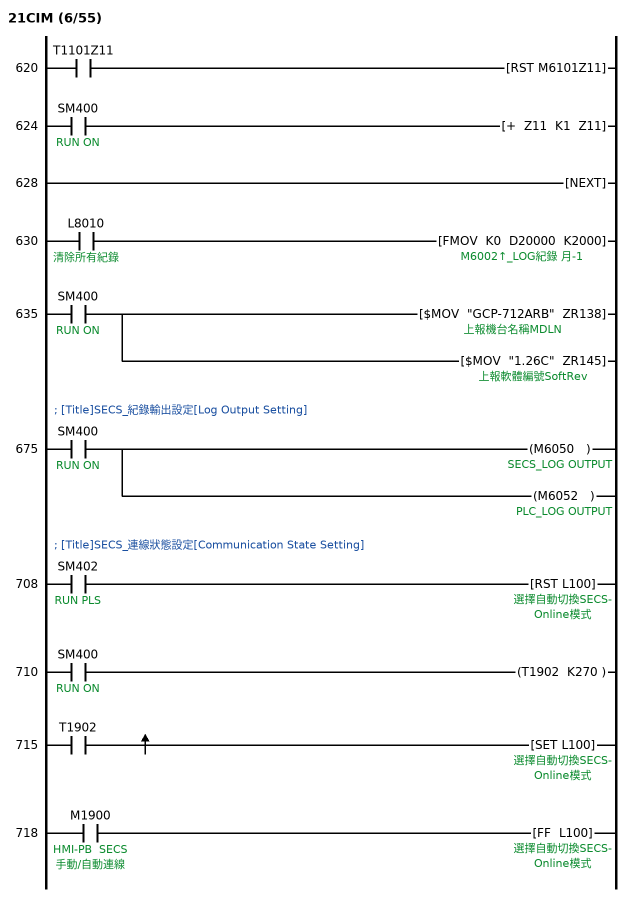
620   LD      T1101Z11
      RST     M6101Z11
624   LD      SM400  ; RUN ON
      +       Z11 K1 Z11
628   NEXT
630   LD      L8010  ; 清除所有紀錄
      FMOV    K0 D20000 K2000  ; M6002↑_LOG紀錄 月-1
635   LD      SM400  ; RUN ON
      $MOV    "GCP-712ARB" ZR138  ; 上報機台名稱MDLN
      $MOV    "1.26C" ZR145  ; 上報軟體編號SoftRev
; [Title]SECS_紀錄輸出設定[Log Output Setting]
675   LD      SM400  ; RUN ON
      OUT     M6050  ; SECS_LOG OUTPUT
      OUT     M6052  ; PLC_LOG OUTPUT
; [Title]SECS_連線狀態設定[Communication State Setting]
708   LD      SM402  ; RUN PLS
      RST     L100  ; 選擇自動切換SECS-Online模式
710   LD      SM400  ; RUN ON
      OUT     T1902 K270
715   LD      T1902
      MEP
      SET     L100  ; 選擇自動切換SECS-Online模式
718   LD      M1900  ; HMI-PB  SECS    手動/自動連線
      FF      L100
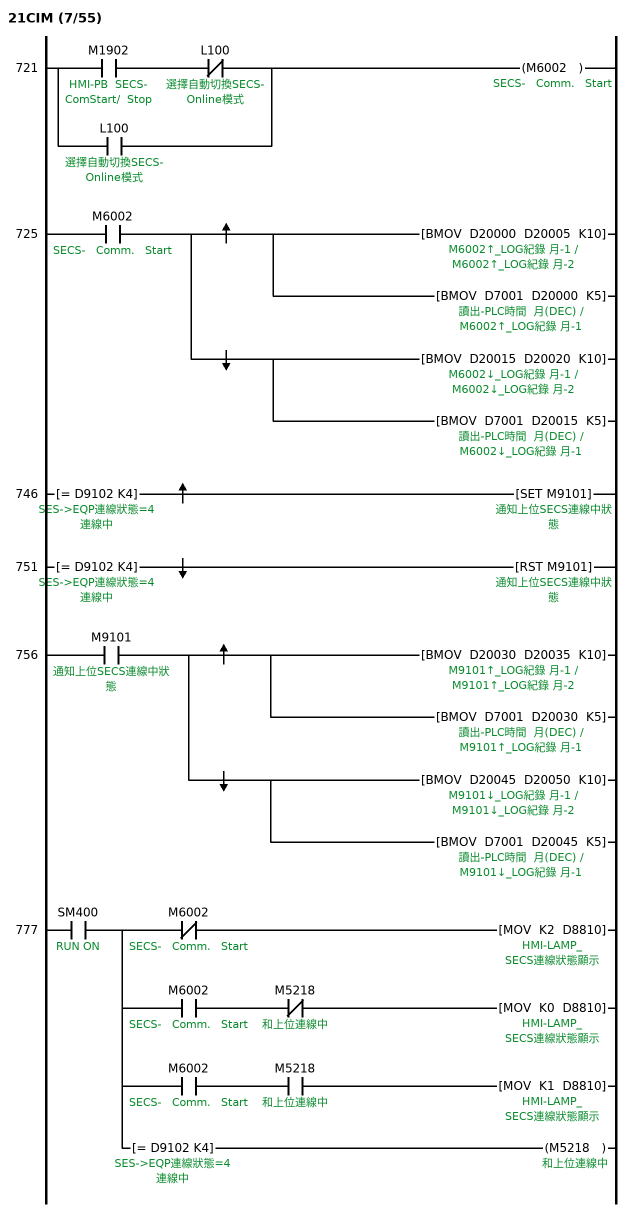
721   LD      M1902  ; HMI-PB  SECS-ComStart/  Stop
      ANI     L100  ; 選擇自動切換SECS-Online模式
      OR      L100  ; 選擇自動切換SECS-Online模式
      OUT     M6002  ; SECS-   Comm.   Start
725   LD      M6002  ; SECS-   Comm.   Start
      MPS
      MEP
      BMOV    D20000 D20005 K10  ; M6002↑_LOG紀錄 月-2
      BMOV    D7001 D20000 K5  ; 讀出-PLC時間  月(DEC)
      MPP
      MEF
      BMOV    D20015 D20020 K10  ; M6002↓_LOG紀錄 月-1 / M6002↓_LOG紀錄 月-2
      BMOV    D7001 D20015 K5
746   LD=     D9102 K4  ; SES->EQP連線狀態=4      連線中
      MEP
      SET     M9101  ; 通知上位SECS連線中狀態
751   LD=     D9102 K4  ; SES->EQP連線狀態=4      連線中
      MEF
      RST     M9101  ; 通知上位SECS連線中狀態
756   LD      M9101  ; 通知上位SECS連線中狀態
      MPS
      MEP
      BMOV    D20030 D20035 K10  ; M9101↑_LOG紀錄 月-1 / M9101↑_LOG紀錄 月-2
      BMOV    D7001 D20030 K5
      MPP
      MEF
      BMOV    D20045 D20050 K10  ; M9101↓_LOG紀錄 月-1 / M9101↓_LOG紀錄 月-2
      BMOV    D7001 D20045 K5
777   LD      SM400  ; RUN ON
      MPS
      ANI     M6002  ; SECS-   Comm.   Start
      MOV     K2 D8810  ; HMI-LAMP_SECS連線狀態顯示
      MRD
      AND     M6002  ; SECS-   Comm.   Start
      ANI     M5218  ; 和上位連線中
      MOV     K0 D8810
      MRD
      AND     M6002  ; SECS-   Comm.   Start
      AND     M5218  ; 和上位連線中
      MOV     K1 D8810
      MPP
      AND=    D9102 K4  ; SES->EQP連線狀態=4      連線中
      OUT     M5218  ; 和上位連線中
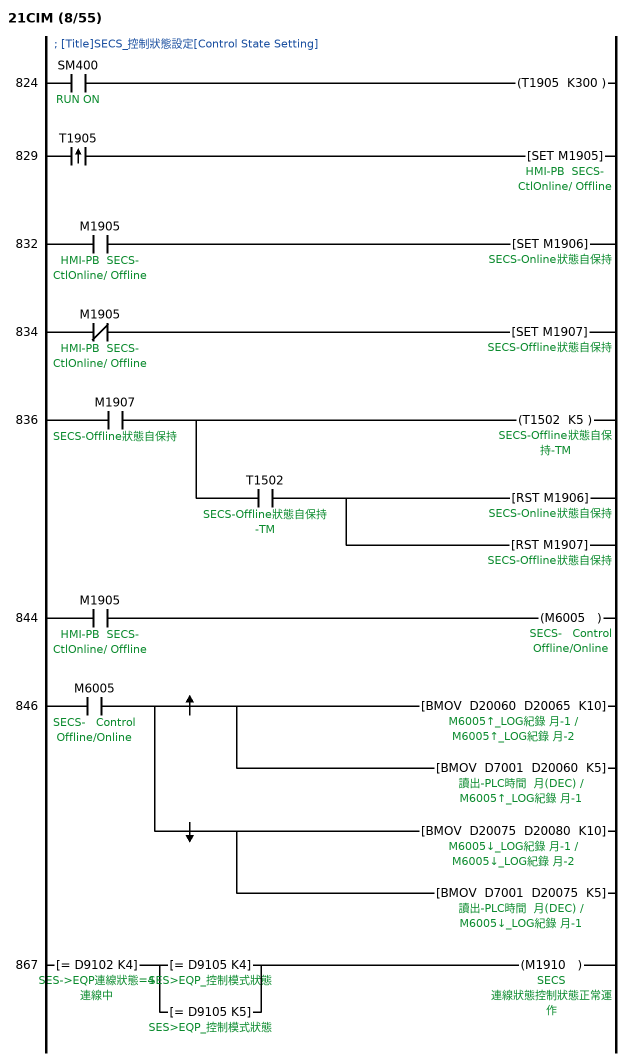
; [Title]SECS_控制狀態設定[Control State Setting]
824   LD      SM400  ; RUN ON
      OUT     T1905 K300
829   LDP     T1905
      SET     M1905  ; HMI-PB  SECS-CtlOnline/ Offline
832   LD      M1905  ; HMI-PB  SECS-CtlOnline/ Offline
      SET     M1906  ; SECS-Online狀態自保持
834   LDI     M1905  ; HMI-PB  SECS-CtlOnline/ Offline
      SET     M1907  ; SECS-Offline狀態自保持
836   LD      M1907  ; SECS-Offline狀態自保持
      OUT     T1502 K5  ; SECS-Offline狀態自保持-TM
      AND     T1502  ; SECS-Offline狀態自保持-TM
      RST     M1906  ; SECS-Online狀態自保持
      RST     M1907  ; SECS-Offline狀態自保持
844   LD      M1905  ; HMI-PB  SECS-CtlOnline/ Offline
      OUT     M6005  ; SECS-   Control Offline/Online
846   LD      M6005  ; SECS-   Control Offline/Online
      MPS
      MEP
      BMOV    D20060 D20065 K10  ; M6005↑_LOG紀錄 月-1 / M6005↑_LOG紀錄 月-2
      BMOV    D7001 D20060 K5
      MPP
      MEF
      BMOV    D20075 D20080 K10  ; M6005↓_LOG紀錄 月-1 / M6005↓_LOG紀錄 月-2
      BMOV    D7001 D20075 K5
867   LD=     D9102 K4  ; SES->EQP連線狀態=4      連線中
      LD=     D9105 K4  ; SES>EQP_控制模式狀態
      OR=     D9105 K5  ; SES>EQP_控制模式狀態
      ANB
      OUT     M1910  ; SECS    連線狀態控制狀態正常運作
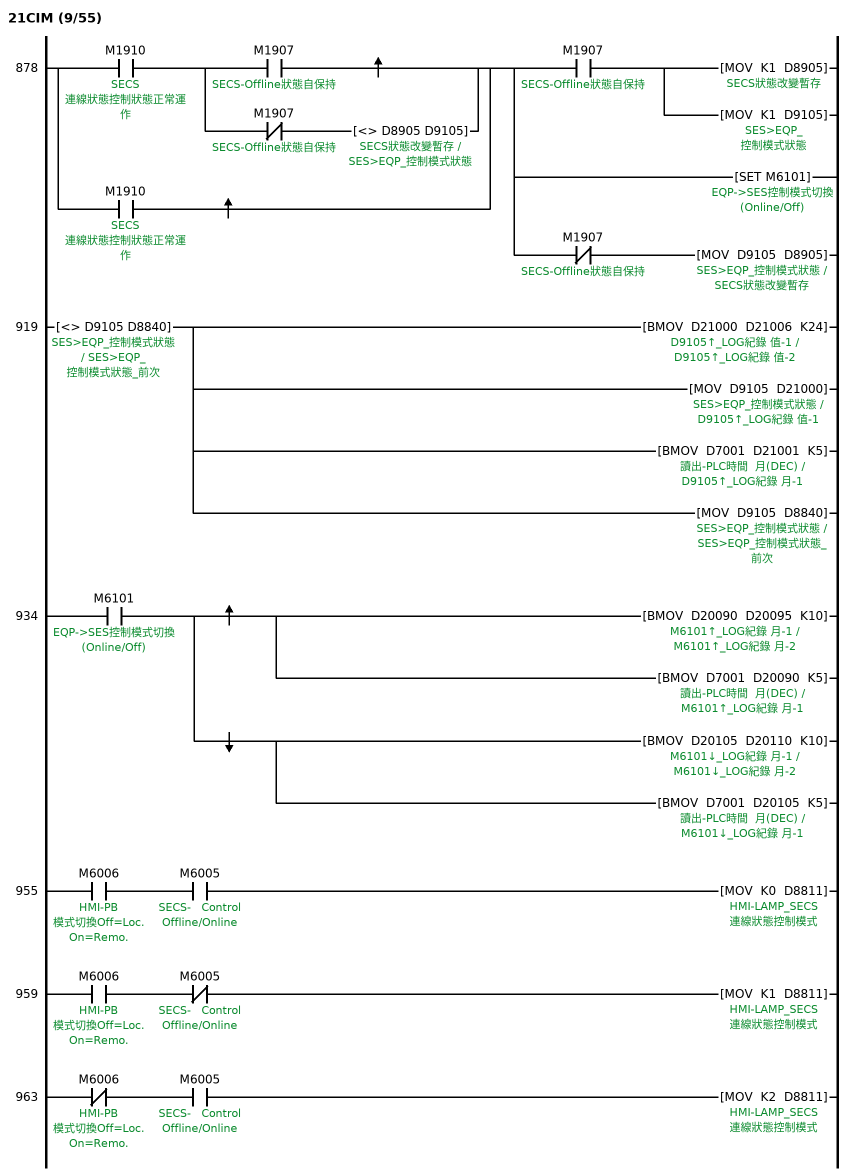
878   LD      M1910  ; SECS    連線狀態控制狀態正常運作
      LD      M1907  ; SECS-Offline狀態自保持
      MEP
      LDI     M1907  ; SECS-Offline狀態自保持
      AND<>   D8905 D9105  ; SECS狀態改變暫存 / SES>EQP_控制模式狀態
      ORB
      ANB
      LD      M1910  ; SECS    連線狀態控制狀態正常運作
      MEP
      ORB
      MPS
      AND     M1907  ; SECS-Offline狀態自保持
      MOV     K1 D8905
        [note] 離線無法上傳狀態，改PLC上報D9105
      MOV     K1 D9105
      MPP
      SET     M6101  ; EQP->SES控制模式切換(Online/Off)
      ANI     M1907  ; SECS-Offline狀態自保持
      MOV     D9105 D8905
919   LD<>    D9105 D8840  ; SES>EQP_控制模式狀態 / SES>EQP_控制模式狀態_前次
      BMOV    D21000 D21006 K24  ; D9105↑_LOG紀錄 值-1 / D9105↑_LOG紀錄 值-2
      MOV     D9105 D21000
      BMOV    D7001 D21001 K5  ; D9105↑_LOG紀錄 月-1
      MOV     D9105 D8840
934   LD      M6101  ; EQP->SES控制模式切換(Online/Off)
      MPS
      MEP
      BMOV    D20090 D20095 K10  ; M6101↑_LOG紀錄 月-1 / M6101↑_LOG紀錄 月-2
      BMOV    D7001 D20090 K5
      MPP
      MEF
      BMOV    D20105 D20110 K10  ; M6101↓_LOG紀錄 月-1 / M6101↓_LOG紀錄 月-2
      BMOV    D7001 D20105 K5
955   LD      M6006  ; HMI-PB  模式切換Off=Loc.On=Remo.
      AND     M6005  ; SECS-   Control Offline/Online
      MOV     K0 D8811  ; HMI-LAMP_SECS   連線狀態控制模式
959   LD      M6006  ; HMI-PB  模式切換Off=Loc.On=Remo.
      ANI     M6005  ; SECS-   Control Offline/Online
      MOV     K1 D8811
963   LDI     M6006  ; HMI-PB  模式切換Off=Loc.On=Remo.
      AND     M6005  ; SECS-   Control Offline/Online
      MOV     K2 D8811
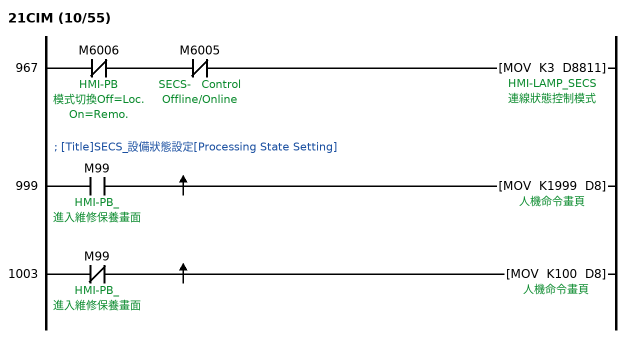
967   LDI     M6006  ; HMI-PB  模式切換Off=Loc.On=Remo.
      ANI     M6005  ; SECS-   Control Offline/Online
      MOV     K3 D8811
; [Title]SECS_設備狀態設定[Processing State Setting]
999   LD      M99  ; HMI-PB_ 進入維修保養畫面
      MEP
      MOV     K1999 D8  ; 人機命令畫頁
1003  LDI     M99  ; HMI-PB_ 進入維修保養畫面
      MEP
      MOV     K100 D8
